FUNCTION_BLOCK MemoOC_D (* CAT Function Block Type *)
  (* Standard: 61499-2 *)
  (* Version 0.0, 6/7/2026, Schneider Electric, template *)
  PACKAGE SE.Nereda;
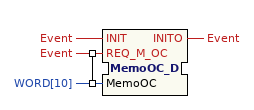
  EVENT_INPUT
    INIT;
    REQ_M_OC WITH MemoOC;
  END_EVENT
  EVENT_OUTPUT
    INITO;
  END_EVENT
  VAR_INPUT
    MemoOC : ARRAY [0..9] OF WORD;
  END_VAR
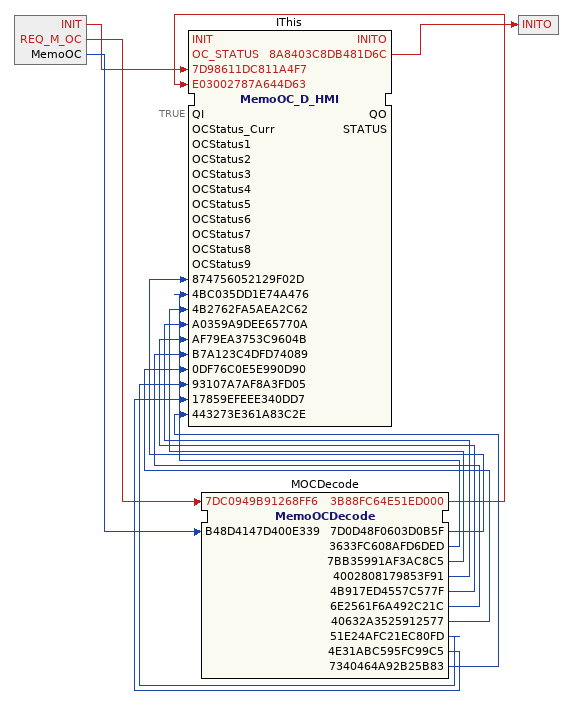
  (* 01 - FUNCTIONNAL INPUT INTERFACE *)
  (* 05 - LOGIC *)
  (* 02 - FUNCTIONNAL OUTPUT INTERFACE *)
  (* 00 - INITIALIZATION *)
  (* 06 - HMI INTERFACE *)
  (* 03 - FIELD INTERFACE *)
  FBS
    IThis : MemoOC_D_HMI(QI := TRUE);
    MOCDecode : MemoOCDecode;
  END_FBS
  EVENT_CONNECTIONS
    INIT TO IThis.7D98611DC811A4F7;
    MOCDecode.3B88FC64E51ED000 TO IThis.E03002787A644D63;
    IThis.8A8403C8DB481D6C TO INITO;
    REQ_M_OC TO MOCDecode.7DC0949B91268FF6;
  END_CONNECTIONS
  DATA_CONNECTIONS
    MOCDecode.7D0D48F0603D0B5F TO IThis.874756052129F02D;
    MOCDecode.3633FC608AFD6DED TO IThis.4BC035DD1E74A476;
    MOCDecode.7BB35991AF3AC8C5 TO IThis.4B2762FA5AEA2C62;
    MOCDecode.4002808179853F91 TO IThis.A0359A9DEE65770A;
    MOCDecode.4B917ED4557C577F TO IThis.AF79EA3753C9604B;
    MOCDecode.6E2561F6A492C21C TO IThis.B7A123C4DFD74089;
    MOCDecode.40632A3525912577 TO IThis.0DF76C0E5E990D90;
    MOCDecode.51E24AFC21EC80FD TO IThis.93107A7AF8A3FD05;
    MOCDecode.4E31ABC595FC99C5 TO IThis.17859EFEEE340DD7;
    MOCDecode.7340464A92B25B83 TO IThis.443273E361A83C2E;
    MemoOC TO MOCDecode.B48D4147D400E339;
  END_CONNECTIONS
END_FUNCTION_BLOCK
